Yaskawa INFORM job: GET-BELOW-POSITION.JBI

/JOB
//NAME GET-BELOW-POSITION
///FOLDERNAME FOLDER001
//POS
///NPOS 0,0,0,4,0,0
///TOOL 1
///POSTYPE ROBOT
///RECTAN
///RCONF 0,0,0,0,0,0,0,0,0,0,0,0,0,0,0,0,0,0,0,0,0,0,0,0
P00094=792.896,160.291,471.972,0.0813,10.0064,0.0684
P00095=1116.664,160.280,463.887,0.0787,10.0067,0.0664
///RCONF 1,0,0,0,0,0,0,0,0,0,0,0,0,0,0,0,0,0,0,0,0,0,0,0
P00124=792.896,161.791,493.972,179.9986,-9.9993,0.0008
P00125=1116.664,160.780,493.887,-179.9993,-9.9981,-0.0025
//INST
///DATE 2025/05/20 21:02
///ATTR SC,RW
///GROUP1 RB1
///LVARS 0,10,20,0,0,0,0,0
NOP
GETE LD001 P125 (1)
GETE LD002 P125 (2)
GETE LD003 P125 (3)
SETE P095 (1) LD001
SETE P095 (2) LD002
SETE P095 (3) LD003
GETE LD001 P124 (1)
GETE LD002 P124 (2)
GETE LD003 P124 (3)
SETE P094 (1) LD001
SETE P094 (2) LD002
SETE P094 (3) LD003
GETE D094 P094 (3)
GETE D095 P095 (3)
ADD D094 -30000
ADD D095 -30000
SETE P094 (3) D094
SETE P095 (3) D095
END
